{attribute addProperty BoxType "EL6201-0000-0017"}
{attribute addProperty Id "Slave_16A_DI0BIT10.125121Slave_16A_DI1BIT10.125122Slave_16A_DI2BIT10.125123Slave_16A_DI3BIT10.125124Slave_16B_DI0BIT10.125125Slave_16B_DI1BIT10.125126Slave_16B_DI2BIT10.125127Slave_16B_DI3BIT10.125128"}
{attribute addProperty CRC "2627028627"}
{attribute addProperty SizeInBites "8"}
{attribute addProperty SizeInBytes "1"}
TYPE Slave_16_Inputs_9C954693 :
STRUCT
	{attribute addProperty Name "Slave_16A_DI0"}
	Slave_16A_DI0 : BIT;
	{attribute addProperty Name "Slave_16A_DI1"}
	Slave_16A_DI1 : BIT;
	{attribute addProperty Name "Slave_16A_DI2"}
	Slave_16A_DI2 : BIT;
	{attribute addProperty Name "Slave_16A_DI3"}
	Slave_16A_DI3 : BIT;
	{attribute addProperty Name "Slave_16B_DI0"}
	Slave_16B_DI0 : BIT;
	{attribute addProperty Name "Slave_16B_DI1"}
	Slave_16B_DI1 : BIT;
	{attribute addProperty Name "Slave_16B_DI2"}
	Slave_16B_DI2 : BIT;
	{attribute addProperty Name "Slave_16B_DI3"}
	Slave_16B_DI3 : BIT;
END_STRUCT
END_TYPE

(* stored: Version 1.2.0.0, ProductVersion 3.1.4024.9
   DUT Slave_16_Inputs_9C954693: Id {0314ca3e-3962-4b1a-94c5-ae059a6b99d7} *)
